(* IEC 61131-3 sources: 2026_Projet_YGO_ExcavatriceDragage/TOOLS/TEST_AUTO_CI/RESULTS/MAIN/tests, 7 files *)

(* ---- test_main_end_to_end.st ---- *)
SETUP
VAR
    mainMachine : FB_Main_EndToEnd;
END_VAR
END_SETUP

TEST 'MAIN_GLOBAL : Chaine Complete - Qualification Neutre vers Montee Treuils Couples'
    // 1. Initialisation boot au neutre (Raw = 5000)
    mainMachine(
        JoyRawX := 5000,
        JoyRawY := 5000,
        JoyDeadmanBtn := FALSE,
        CmdMode := E_Mode.MAINT_N1,
        CmdWinchSelect := 1,
        EmergencyChainClosed := TRUE,
        PowerContactorEngaged := TRUE
    );
    mainMachine(
        JoyRawX := 5000,
        JoyRawY := 5000,
        JoyDeadmanBtn := TRUE, // Début appui homme-mort au neutre
        CmdMode := E_Mode.MAINT_N1,
        CmdWinchSelect := 1,
        EmergencyChainClosed := TRUE,
        PowerContactorEngaged := TRUE
    );
    ADVANCE_TIME(150000000); // 150 ms (> 100 ms DeadmanArmHoldTime)
    mainMachine(
        JoyRawX := 5000,
        JoyRawY := 5000,
        JoyDeadmanBtn := TRUE, // Confirmation maintien homme-mort -> Armé
        CmdMode := E_Mode.MAINT_N1,
        CmdWinchSelect := 1,
        EmergencyChainClosed := TRUE,
        PowerContactorEngaged := TRUE
    );

    // 2. Stimulus Opérateur : Poussée Manche vers le Haut (+Y = 8000) avec Homme-mort maintenu
    mainMachine(
        JoyRawX := 5000,
        JoyRawY := 8000, // Déviation Y Montée
        JoyDeadmanBtn := TRUE,
        CmdMode := E_Mode.MAINT_N1,
        CmdWinchSelect := 1,
        EmergencyChainClosed := TRUE,
        PowerContactorEngaged := TRUE
    );
    mainMachine(
        JoyRawX := 5000,
        JoyRawY := 8000,
        JoyDeadmanBtn := TRUE,
        CmdMode := E_Mode.MAINT_N1,
        CmdWinchSelect := 1,
        EmergencyChainClosed := TRUE,
        PowerContactorEngaged := TRUE
    );

    // 3. Vérification des flux à travers toute la machine (PRG_02 -> PRG_07)
    // - Bus PRG_02 : Joystick armé et qualifié
    ASSERT_TRUE(mainMachine.BusAcq.JoystickDeadmanArmed, 'PRG_02: Homme-mort qualifie');

    // - Bus PRG_03 : Mode Manuel N1 arbitré
    ASSERT_EQ(mainMachine.BusModes.Mode, E_Mode.MAINT_N1, 'PRG_03: Mode MAINT_N1 arbitre');

    // - Bus PRG_04 : Demande de montée et sécurité nominale
    ASSERT_FALSE(mainMachine.BusWinch.WinchM1Safety.SafeStop, 'PRG_04: Aucun SafeStop actif');

    // - Bus PRG_07 : Bandeau IHM informé sans défaut
    ASSERT_TRUE(mainMachine.BusBanner.GlobalContextText <> '', 'PRG_07: Bandeau IHM present');
    ASSERT_FALSE(mainMachine.BusBanner.AlarmBanner.HasAlarm, 'PRG_07: Aucune alarme bloqueuse');
END_TEST

TEST 'MAIN_GLOBAL : Coupure Puissance AU Propagee a tous les Actionneurs'
    // Stimulus : Chute de la boucle AU physique
    mainMachine(
        JoyRawX := 0,
        JoyRawY := 1000,
        JoyDeadmanBtn := TRUE,
        CmdMode := E_Mode.MAINT_N1,
        EmergencyChainClosed := FALSE, // Chaîne AU ouverte
        PowerContactorEngaged := FALSE
    );

    // Vérification : toutes les sorties physiques sont instantanément coupées
    ASSERT_FALSE(mainMachine.BusOutputs.M1RelayFwd, 'Coupure immediate relais M1');
    ASSERT_FALSE(mainMachine.BusOutputs.M1BrakeCmd, 'Frein M1 retombe');
    ASSERT_FALSE(mainMachine.BusOutputs.TranslationBrakeCmd, 'Frein M3 bloque');
END_TEST

(* ---- test_prg_02_acquisition.st ---- *)
SETUP
VAR
    harness : FB_TestHarness_PRG_02;
END_VAR
END_SETUP

TEST 'PRG_02_Acquisition : Qualification joystick (neutre -> armement -> consigne X)'
    // 1. Initialisation au neutre
    harness(JoyRawX := 5000, JoyRawY := 5000, JoyBtnRaw := FALSE);
    ADVANCE_TIME(60000000);
    harness(JoyRawX := 5000, JoyRawY := 5000, JoyBtnRaw := TRUE); // Appui homme-mort au neutre
    ADVANCE_TIME(60000000);
    harness(JoyRawX := 5000, JoyRawY := 5000, JoyBtnRaw := TRUE);
    ASSERT_TRUE(harness.Data.JoystickDeadmanArmed, 'Homme-mort arme avec succes');

    // 2. Mouvement manche a droite (RawX = 8000)
    harness(JoyRawX := 8000, JoyRawY := 5000, JoyBtnRaw := FALSE);
    ASSERT_EQ(harness.Data.JoystickDirectionX, 1, 'Sens X positif detecte (Translation Droite)');
    ASSERT_GT(harness.Data.JoystickSpeedPctX, 0.0, 'Consigne de vitesse non nulle transmise sur le bus Data');
END_TEST

TEST 'PRG_02_Acquisition : Decodage capteurs Translation M3 et calcul mot de position'
    // Activation capteurs zone Tremie (SensorTremie=TRUE, SensorPV=TRUE, SensorP2=TRUE, SensorP1=TRUE, SensorMaintenance=TRUE -> 2#11111)
    harness(
        M3_PosTremie_DI := TRUE,
        M3_PosPV_DI := TRUE,
        M3_PosPVP2_DI := TRUE,
        M3_PosP1_DI := TRUE,
        M3_PosMaintenance_DI := TRUE
    );
    ASSERT_TRUE(harness.Data.TranslationAtTremie, 'Position exacte Tremie atteinte');
    ASSERT_TRUE(harness.Data.M3_LimitSwitchFwd, 'Fin de course avant actif a la tremie');
    ASSERT_FALSE(harness.Data.M3_SensorWordIncoherent, 'Mot capteurs coherent');
END_TEST

(* ---- test_prg_03_modes_cycle.st ---- *)
SETUP
VAR
    harness : FB_TestHarness_PRG_03;
END_VAR
END_SETUP

TEST 'PRG_03_Modes_Cycle : Mode Manuel MAINT_N1 (autorisations unitaires et arbitrage)'
    harness(
        SelMode := E_Mode.MAINT_N1,
        PowerContactorEngaged := TRUE,
        SelJoystickWinch := 1 // M1
    );
    ASSERT_EQ(harness.Auth.Mode, E_Mode.MAINT_N1, 'Mode MAINT_N1 arbitre');
    ASSERT_EQ(harness.Auth.JoystickWinchSelectArbitrated, 1, 'Selection Joystick M1 arbitree');
    ASSERT_FALSE(harness.Auth.InhibitM1, 'Inhibition M1 interdite en N1');
END_TEST

TEST 'PRG_03_Modes_Cycle : Mode Semi-Auto (activation sequenceur et etape initiale)'
    harness(
        SelMode := E_Mode.SEMI_AUTO,
        PowerContactorEngaged := TRUE,
        HomedM1 := TRUE,
        HomedM2 := TRUE
    );
    ASSERT_EQ(harness.Auth.Mode, E_Mode.SEMI_AUTO, 'Mode SEMI_AUTO arbitre');
    ASSERT_EQ(harness.CycleStep, E_CycleStep.X0_PREPARATION, 'Sequenceur pret a l etape X0_PREPARATION');
END_TEST

(* ---- test_prg_04_treuils_benne.st ---- *)
SETUP
VAR
    harness : FB_TestHarness_PRG_04;
    acqData : ST_AcquisitionInterPrg;
    modesAuth : ST_Modes_Autorisations;
END_VAR
END_SETUP

TEST 'PRG_04_Treuils_Benne : Commande Montee M1 via Bus AcqData + ModesAuth'
    // 1. Contexte : Mode Manuel N1, Treuil M1 selectionne
    modesAuth.Mode := E_Mode.MAINT_N1;
    modesAuth.JoystickWinchSelectArbitrated := 1; // M1

    // 2. Stimulus issu du bus PRG_02 : Homme mort arme, manche non centre (Montee)
    acqData.JoystickDeadmanArmed := TRUE;
    acqData.JoystickYNeutral := FALSE;
    acqData.JoystickDirectionX := 0;
    acqData.CablePosM1 := 2.0;
    acqData.M1_Speed_Mps := 0.0;

    // 3. Execution PRG_04 (2 cycles pour passer le premier scan d'init FirstScanDone)
    harness(
        AcqData := acqData,
        ModesAuth := modesAuth,
        BtnWinchM1Up := TRUE,
        PowerContactorEngaged := TRUE,
        M1_ContactorsReleased := TRUE
    );
    harness(
        AcqData := acqData,
        ModesAuth := modesAuth,
        BtnWinchM1Up := TRUE,
        PowerContactorEngaged := TRUE,
        M1_ContactorsReleased := TRUE
    );

    // 4. Verification des demandes produites sur le bus sortant ST_WinchInterPrg
    ASSERT_TRUE(harness.Data.WinchM1FinalInterlockRequest.RequestedRelayFwd, 'Ordre RelayFwd genere vers PRG_06');
    ASSERT_FALSE(harness.Data.WinchM1Safety.SafeStop, 'Aucun SafeStop actif');
END_TEST

TEST 'PRG_04_Treuils_Benne : SafeStop Treuil M1 sur Defaut Codeur'
    // Stimulus : Defaut codeur remonte par le bus PRG_02
    acqData.M1_EncoderFault := TRUE;

    harness(
        AcqData := acqData,
        ModesAuth := modesAuth,
        PowerContactorEngaged := TRUE
    );

    ASSERT_TRUE(harness.Data.WinchM1Safety.SafeStop, 'SafeStop declenche immediatement sur defaut codeur');
    ASSERT_FALSE(harness.Data.WinchM1FinalInterlockRequest.RequestedRelayFwd, 'Mouvement neutralise');
END_TEST

(* ---- test_prg_05_translation.st ---- *)
SETUP
VAR
    harness   : FB_TestHarness_PRG_05;
    acqData   : ST_AcquisitionInterPrg;
    modesAuth : ST_Modes_Autorisations;
END_VAR
END_SETUP

TEST 'PRG_05_Translation : Commande Translation Fwd (Joystick X + Hauteur Treuils OK)'
    // 1. Contexte : Mode Manuel N1, Câbles treuils hauts (sécurité interlock hauteur validée)
    modesAuth.Mode := E_Mode.MAINT_N1;

    // 2. Stimulus issu du bus PRG_02 : Joystick armé vers la droite (+X)
    acqData.JoystickDeadmanArmed := TRUE;
    acqData.JoystickDirectionX := 1;
    acqData.JoystickSpeedPctX := 75.0;
    acqData.M3_LimitSwitchFwd := FALSE; // Non en butée
    acqData.M3_LimitSwitchRev := FALSE;
    acqData.TranslationAtPV := FALSE;
    acqData.TranslationAtP1 := FALSE;
    acqData.TranslationAtP2 := FALSE;

    // 3. Exécution PRG_05 (3 scans : 1=FirstScanDone, 2=CommandedDirection, 3=SpeedRamp/Brake)
    harness(
        AcqData := acqData,
        ModesAuth := modesAuth,
        WinchM1CablePosM := 5.0,
        WinchM2CablePosM := 5.0,
        PowerContactorEngaged := TRUE,
        DriveOnline := TRUE,
        DriveOperational := TRUE
    );
    harness(
        AcqData := acqData,
        ModesAuth := modesAuth,
        WinchM1CablePosM := 5.0,
        WinchM2CablePosM := 5.0,
        PowerContactorEngaged := TRUE,
        DriveOnline := TRUE,
        DriveOperational := TRUE
    );
    harness(
        AcqData := acqData,
        ModesAuth := modesAuth,
        WinchM1CablePosM := 5.0,
        WinchM2CablePosM := 5.0,
        PowerContactorEngaged := TRUE,
        DriveOnline := TRUE,
        DriveOperational := TRUE
    );

    // 4. Vérification du bus sortant ST_TranslationInterPrg vers PRG_06
    ASSERT_TRUE(harness.Data.TranslationFinalInterlockRequest.BrakeReleaseRequest, 'Demande desserrage frein M3 generee');
    ASSERT_FALSE(harness.Data.TranslationSafety.SafeStop, 'Aucun SafeStop actif sur translation');
    ASSERT_EQ(harness.Data.TranslationState.ActiveDirection, 1, 'Sens translation avant arbitre');
END_TEST

TEST 'PRG_05_Translation : Interdiction Mouvement Translation si Treuils en Bas'
    // Stimulus : Treuil M1 descendu trop bas (< 2m)
    harness(
        AcqData := acqData,
        ModesAuth := modesAuth,
        WinchM1CablePosM := 0.5,
        WinchM2CablePosM := 5.0,
        PowerContactorEngaged := TRUE
    );

    // Vérification : mouvement bloqué par l'interlock de hauteur
    ASSERT_FALSE(harness.Data.TranslationFinalInterlockRequest.BrakeReleaseRequest, 'Frein reste serre');
    ASSERT_EQ(harness.Data.TranslationState.ActiveDirection, 0, 'Mouvement interdit');
END_TEST

(* ---- test_prg_06_outputs.st ---- *)
SETUP
VAR
    harness         : FB_TestHarness_PRG_06;
    winchData       : ST_WinchInterPrg;
    translationData : ST_TranslationInterPrg;
END_VAR
END_SETUP

TEST 'PRG_06_Outputs : Transmission Ordres M1 et M3 en Marche Normale'
    // 1. Contexte M1 : Demande de montée active avec contacteur 1
    winchData.WinchM1FinalInterlockRequest.Enable := TRUE;
    winchData.WinchM1FinalInterlockRequest.PowerContactorEngaged := TRUE;
    winchData.WinchM1FinalInterlockRequest.SafeStop := FALSE;
    winchData.WinchM1FinalInterlockRequest.PowerCutOff := FALSE;
    winchData.WinchM1FinalInterlockRequest.RequestedRelayFwd := TRUE;
    winchData.WinchM1FinalInterlockRequest.RequestedContactor1 := TRUE;
    winchData.WinchM1FinalInterlockRequest.RequestedStep := 1;
    winchData.WinchM1FinalInterlockRequest.FwdRevSpeedFeedbackOff := TRUE;

    // 2. Contexte M3 : Demande de frein relâché
    translationData.TranslationFinalInterlockRequest.Enable := TRUE;
    translationData.TranslationFinalInterlockRequest.PowerContactorEngaged := TRUE;
    translationData.TranslationFinalInterlockRequest.SafeStop := FALSE;
    translationData.TranslationFinalInterlockRequest.PowerCutOff := FALSE;
    translationData.TranslationFinalInterlockRequest.BrakeReleaseRequest := TRUE;

    // 3. Exécution PRG_06
    harness(
        WinchData := winchData,
        TranslationData := translationData
    );

    // 4. Vérification des sorties réelles sur le bus ST_OutputsInterPrg
    ASSERT_TRUE(harness.Data.M1RelayFwd, 'Contacteur montee M1 active');
    ASSERT_TRUE(harness.Data.M1SpeedContactor1, 'Palier 1 M1 active');
    ASSERT_TRUE(harness.Data.M1BrakeCmd, 'Commande desserrage frein M1 active');
    ASSERT_TRUE(harness.Data.TranslationBrakeCmd, 'Commande desserrage frein M3 active');
END_TEST

TEST 'PRG_06_Outputs : Barriere de Securite Coupure Brutale PowerCutOff sur M1'
    // Stimulus : Demande de montée avec PowerCutOff actif sur M1
    winchData.WinchM1FinalInterlockRequest.PowerCutOff := TRUE;

    harness(
        WinchData := winchData,
        TranslationData := translationData
    );

    // Vérification : toutes les sorties M1 doivent être immédiatement neutralisées
    ASSERT_FALSE(harness.Data.M1RelayFwd, 'Relais montee M1 coupe');
    ASSERT_FALSE(harness.Data.M1SpeedContactor1, 'Contacteurs vitesse M1 coupes');
    ASSERT_FALSE(harness.Data.M1BrakeCmd, 'Frein M1 retombe');
END_TEST

(* ---- test_prg_07_supervision.st ---- *)
SETUP
VAR
    harness         : FB_TestHarness_PRG_07;
    acqData         : ST_AcquisitionInterPrg;
    modesAuth       : ST_Modes_Autorisations;
    winchData       : ST_WinchInterPrg;
    translationData : ST_TranslationInterPrg;
END_VAR
END_SETUP

TEST 'PRG_07_Supervision : Formatage Bandeau IHM Mode Manuel Sans Defaut'
    // 1. Contexte : Mode Manuel N1
    modesAuth.Mode := E_Mode.MAINT_N1;
    modesAuth.JoystickWinchSelectArbitrated := 0; // Couplé

    // 2. Stimulus : Machine saine, puissance engagée
    acqData.JoystickDeadmanArmed := TRUE;
    acqData.JoystickYNeutral := TRUE;
    winchData.WinchM1Safety.DescendPermit := TRUE;
    winchData.WinchM1Safety.AscentPermit := TRUE;
    winchData.WinchM2Safety.DescendPermit := TRUE;
    winchData.WinchM2Safety.AscentPermit := TRUE;

    // 3. Exécution PRG_07
    harness(
        AcqData := acqData,
        ModesAuth := modesAuth,
        WinchData := winchData,
        TranslationData := translationData,
        PowerContactorEngaged := TRUE,
        EmergencyChainClosed := TRUE,
        PowerCutOffActive := FALSE
    );

    // 4. Vérification de la présence d'un bandeau IHM cohérent
    ASSERT_TRUE(harness.Banner.GlobalContextText <> '', 'Contexte global IHM renseigne');
END_TEST

TEST 'PRG_07_Supervision : Remontee Alarme Bandeau sur SafeStop Treuil'
    // Stimulus : SafeStop actif sur Treuil M1 avec défaut codeur
    winchData.WinchM1Safety.SafeStop := TRUE;
    winchData.WinchM1Safety.Error := TRUE;
    winchData.WinchM1Safety.ErrorEncoder := TRUE;
    winchData.WinchM1Safety.ErrorId := 16#0002; // Perte codeur

    harness(
        AcqData := acqData,
        ModesAuth := modesAuth,
        WinchData := winchData,
        TranslationData := translationData,
        PowerContactorEngaged := TRUE
    );

    // Vérification de la notification d'alarme dans le bandeau
    ASSERT_TRUE(harness.Banner.AlarmBanner.HasAlarm, 'Alarme active visible sur le bandeau IHM');
END_TEST
